{attribute 'pack_mode' := '1'}
TYPE ST_TxCanQueue_29bit_CX2500_M510 :
STRUCT
	nTxCounter: UINT; 		// Tx Handshake
	nRxCounter: UINT; 		// Rx handshake
	nNoOfmessages: UINT; 	// Number of messages relevent in Queue, ignore the rest.
	nDummy : UINT;			//Reserved
	aMessages: ARRAY[0..GVL_CanItfHelper.nTxQueueUpperIndex] OF ST_CanData_29bit_CX2500_M510;
END_STRUCT
END_TYPE

(* stored: Version 1.1.0.1, ProductVersion 3.1.4024.12
   DUT ST_TxCanQueue_29bit_CX2500_M510: Id {835ee193-80ef-0351-0b9d-edb5e21331e1} *)
